{attribute 'qualified_only'}
{attribute 'to_string'}
// Fault codes surfaced by FB_StateMachine through ST_DeviceHeader_Sts (the
// fault book-keeping lives on FB_DeviceBase). Range convention mirrors
// E_RpcMethodResponse so codes are self-documenting:
//
//   0        No fault
//   1-9      Timeouts
//   10-19    Feedback / hardware
//   20-29    State violations
//   30-39    Configuration
//   50-59    Interlocks / permissives
//   70-79    Submodule / propagation
//   100+     Device / application custom
//
// HMI displays ResolveFaultString(code) for the stable title and faultReason
// for the contextual detail (step number, step name, free-form operator
// message). Both live in ST_DeviceHeader_Sts.
TYPE E_SM_Fault :
(
    None                    := 0,

    StepTimeout             := 1,    // FB_Step.tonTimeout expired
    OddStepReached          := 2,    // default fault when a step moves onto an odd step number
    StepUserFault           := 3,    // user called step.RaiseFault(code, reason)

    InvalidStepConfiguration := 30,
    MissingStepImplementation := 31,
    DuplicateStepImplementation := 32,
    ShutdownFailed := 33,

    RunningInterlockTripped := 50,   // intlkRunning tripped, auto-aborted

    SubmoduleFaulted        := 70    // external inpSubmoduleFaulted asserted
);
END_TYPE

(* stored: Version 1.1.0.1, ProductVersion 3.1.4026.12
   DUT E_SM_Fault: Id {a1b2c3d4-0002-0001-0001-000000000001} *)
